(* Logix 5000 project; controller APM_EXTRUSORA Emulate 5570 rev 30.12; software revision 30.00 *)

TASK MainTask (continuous, watchdog 500 ms) : MainProgram

MODULES
   Local : Emulate 5570 (ICP 2, rev 30.12)
      VIRTUAL_OUTPUTS : vendor 1 type 0 code 15 (ICP 4, rev 1.1, Output RPI 50 ms)
      VIRTUAL_INPUTS : vendor 1 type 0 code 15 (ICP 3, rev 1.1, Output RPI 50 ms)
END_MODULES

VAR_GLOBAL   (* controller tags *)
   START : ALIAS FOR Local:3:I.Data[1].0;
   STARTED : ALIAS FOR Local:4:O.Data[0].0;
   STOP : ALIAS FOR Local:3:I.Data[1].1;
   Temporizador_Plastico : TIMER := (PRE := 8000);   // Cuenta cada cuanto tiempo se debe liberar lástico en la extrución
   TON_EP2 : TIMER := (PRE := 300);   // Da una leve espera para reiniciar el Temporizador_Plastico
END_VAR

PROGRAM MainProgram   (* main routine MainRoutine *)

ROUTINE MainRoutine   (* ladder *)
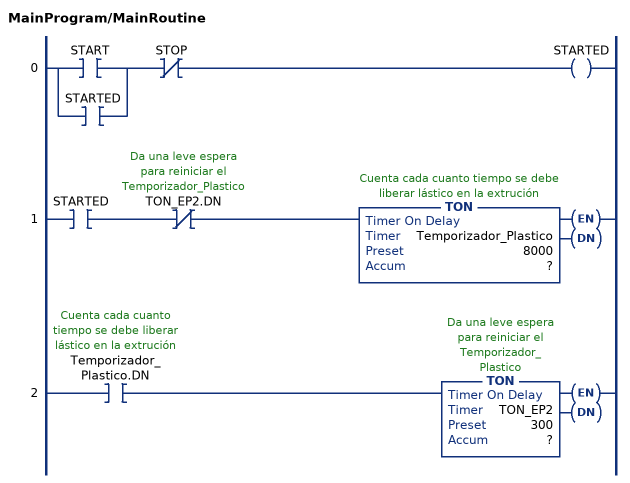
   0: [XIC(START) ,XIC(STARTED) ]XIO(STOP)OTE(STARTED);
   1: XIC(STARTED)XIO(TON_EP2.DN)TON(Temporizador_Plastico,?,?);
   2: XIC(Temporizador_Plastico.DN)TON(TON_EP2,?,?);
END_ROUTINE
END_PROGRAM
